FUNCTION_BLOCK FB_Integer_To_BooleanArray
VAR_INPUT
	IntegerValue: INT := -1; // Int value from RadioButton or whatever indexed component
	ArrayLength: INT := 2; // rquired length of the output Array 
END_VAR
VAR_OUTPUT
	OutputValue: ARRAY [0..1] OF BOOL; 
END_VAR
VAR
	i: INT;  // Loop counter
END_VAR



FOR i := 0 TO (ArrayLength -1) DO
    OutputValue[i] := (IntegerValue = i);    // Set the corresponding boolean value based on the radiobutton value
END_FOR

END_FUNCTION_BLOCK

(* stored: Version 1.1.0.1, ProductVersion 3.1.4024.12
   POU FB_Integer_To_BooleanArray: Id {acd2210e-3c7d-46ac-a1a0-7ba37313b6e6}, SpecialFunc None *)
